TYPE E_MeasureOption :
(
	MEAS_OPTION_SlowApproach := 0,
	MEAS_OPTION_FastApproach := 1,
	MEAS_OPTION_OnlyXY := 2
)USINT;
END_TYPE

(* stored: Version 1.1.0.1, ProductVersion 3.1.0.25
   DUT E_MeasureOption: Id {bd9d8bd6-02ed-4764-bb46-2b338e63c7ec} *)
